{attribute 'hide'}
FUNCTION_BLOCK FileSystemEntryCollection_Test EXTENDS TcUnit.FB_TestSuite

CountReturnsZeroAfterClear();
CountReturnsExpectedAfterInsert();
GetFirstReturnsNullIfEmpty();
GetNextReturnsNullIfEmpty();
GetFirstReturnsExpected();
GetNextReturnsExpected();

METHOD CountReturnsExpectedAfterInsert
VAR
	collection : FileSystemEntryCollection;
	mockFileSystemEntry : Mock_FilesystemEntry('');
	expected : INT;
	actual : INT;
END_VAR
TEST('CountReturnsExpectedAfterInsert');

// @TEST-FIXTURE
expected := 2;

// @TEST-RUN
collection.Insert(mockFileSystemEntry);
collection.Insert(mockFileSystemEntry);
actual := collection.Count;

// @TEST-ASSSERT
AssertEquals_INT(Expected := expected, Actual := actual, Message := 'Count did not return expected');

TEST_FINISHED();
END_METHOD

METHOD CountReturnsZeroAfterClear
VAR
	collection : FileSystemEntryCollection;
	expected : INT;
	actual : INT;
END_VAR
TEST('CountReturnsZeroAfterClear');

// @TEST-FIXTURE
expected := 0;

// @TEST-RUN
collection.Clear();
actual := collection.Count;

// @TEST-ASSSERT
AssertEquals_INT(Expected := expected, Actual := actual, Message := 'Count did not return zero');

TEST_FINISHED();
END_METHOD

METHOD GetByIndexReturnsExpected
VAR
	collection : FileSystemEntryCollection;
	mockFileSystemEntry1 : Mock_FilesystemEntry('C:\TestPath_1\');
	mockFileSystemEntry2 : Mock_FilesystemEntry('C:\TestPath_2\');
	entry : I_FileSystemEntry;
	expected : FilePath;
	actual : FilePath;
END_VAR
TEST('GetByIndexReturnsExpected');

// @TEST-FIXTURE
expected := 'C:\TestPath_2\';

// @TEST-RUN
collection.Insert(mockFileSystemEntry1);
collection.Insert(mockFileSystemEntry2);
entry := collection.GetByIndex(1);


actual := entry.Path;

// @TEST-ASSSERT
AssertEquals_STRING(Expected := expected, Actual := actual, Message := 'Did not return expected');

TEST_FINISHED();
END_METHOD

METHOD GetByIndexReturnsNullIfEmpty
VAR
	collection : FileSystemEntryCollection;
	entry : I_FileSystemEntry;
	result : BOOL;
END_VAR
TEST('GetByIndexReturnsNullIfEmpty');

// @TEST-FIXTURE

// @TEST-RUN
collection.Clear();
entry := collection.GetByIndex(0);
result := entry.IsNull;

// @TEST-ASSSERT
AssertTrue(Condition := result, Message := 'Did not return a null entry');

TEST_FINISHED();
END_METHOD

METHOD GetByIndexReturnsNullIfIndexOutOfRange
VAR
	collection : FileSystemEntryCollection;
	entry1 : I_FileSystemEntry;
	entry2 : I_FileSystemEntry;
	result1 : BOOL;
	result2 : BOOL;
END_VAR
TEST('GetByIndexReturnsNullIfIndexOutOfRange');

// @TEST-FIXTURE

// @TEST-RUN
collection.Clear();
entry1 := collection.GetByIndex(-1);
entry2 := collection.GetByIndex(100);
result1 := entry1.IsNull;
result2 := entry2.IsNull;


// @TEST-ASSSERT
AssertTrue(Condition := result1, Message := 'Did not return a null entry');
AssertTrue(Condition := result2, Message := 'Did not return a null entry');

TEST_FINISHED();
END_METHOD

METHOD GetFirstReturnsExpected
VAR
	collection : FileSystemEntryCollection;
	mockFileSystemEntry : Mock_FilesystemEntry('C:\TestPath\');
	entry : I_FileSystemEntry;
	expected : FilePath;
	actual : FilePath;
END_VAR
TEST('GetFirstReturnsExpected');

// @TEST-FIXTURE
expected := 'C:\TestPath\';

// @TEST-RUN
collection.Insert(mockFileSystemEntry);
entry := collection.GetFirst();

actual := entry.Path;

// @TEST-ASSSERT
AssertEquals_STRING(Expected := expected, Actual := actual, Message := 'Did not return expected');

TEST_FINISHED();
END_METHOD

METHOD GetFirstReturnsNullIfEmpty
VAR
	collection : FileSystemEntryCollection;
	entry : I_FileSystemEntry;
	result : BOOL;
END_VAR
TEST('GetFirstReturnsNullIfEmpty');

// @TEST-FIXTURE

// @TEST-RUN
collection.Clear();
entry := collection.GetFirst();
result := entry.IsNull;

// @TEST-ASSSERT
AssertTrue(Condition := result, Message := 'Did not return a null entry');

TEST_FINISHED();
END_METHOD

METHOD GetNextReturnsExpected
VAR
	collection : FileSystemEntryCollection;
	mockFileSystemEntry1 : Mock_FilesystemEntry('C:\TestPath_1\');
	mockFileSystemEntry2 : Mock_FilesystemEntry('C:\TestPath_2\');
	entry : I_FileSystemEntry;
	expected : FilePath;
	actual : FilePath;
END_VAR
TEST('GetNextReturnsExpected');

// @TEST-FIXTURE
expected := 'C:\TestPath_2\';

// @TEST-RUN
collection.Insert(mockFileSystemEntry1);
collection.Insert(mockFileSystemEntry2);
entry := collection.GetFirst();
entry := collection.GetNext(entry);

actual := entry.Path;

// @TEST-ASSSERT
AssertEquals_STRING(Expected := expected, Actual := actual, Message := 'Did not return expected');

TEST_FINISHED();
END_METHOD

METHOD GetNextReturnsNullIfEmpty
VAR
	collection : FileSystemEntryCollection;
	entry : I_FileSystemEntry;
	result : BOOL;
END_VAR
TEST('GetNextReturnsNullIfEmpty');

// @TEST-FIXTURE

// @TEST-RUN
collection.Clear();
entry := collection.GetNext(0);
result := entry.IsNull;

// @TEST-ASSSERT
AssertTrue(Condition := result, Message := 'Did not return a null entry');

TEST_FINISHED();
END_METHOD

END_FUNCTION_BLOCK

(* stored: Version 1.1.0.1, ProductVersion 3.1.4024.9
   POU FileSystemEntryCollection_Test: Id {2c9e117c-3f29-4d88-acd3-30a0f57a34d9}, SpecialFunc None
   Method CountReturnsExpectedAfterInsert: Id {78cd8310-e4e5-4401-aee5-e86d1a558e63}
   Method CountReturnsZeroAfterClear: Id {e625bb33-48a7-4c4e-95a9-9ba35fc2f5a8}
   Method GetByIndexReturnsExpected: Id {88c77a78-6131-4253-92a6-9ac95ffbd296}
   Method GetByIndexReturnsNullIfEmpty: Id {c3de5e3a-10a6-4e78-ab45-5eb4e12732b1}
   Method GetByIndexReturnsNullIfIndexOutOfRange: Id {50318e51-651f-4eed-8cca-fcf06a57fd5d}
   Method GetFirstReturnsExpected: Id {c49a26a0-04bc-4fc3-bbc7-9450dfbba9db}
   Method GetFirstReturnsNullIfEmpty: Id {c8f80720-ad8a-4597-952d-b8ba38004345}
   Method GetNextReturnsExpected: Id {587a45c8-c3f7-4bfc-ad57-3491a6be1142}
   Method GetNextReturnsNullIfEmpty: Id {7a3fe986-d18b-46ab-943f-d09713213fa5} *)
